Omron CX-Programmer project NewProject (CX-Programmer 9.81)

# PLC Sessao_10_02_2026_Exercicios: CP1L-E EM

## Global symbols (name address type ; comment)
0.00 BOOL  ; Interuptor 1
0.01 BOOL  ; Interruptor 2
0.02 BOOL  ; Botao de Emergencia
0.03 BOOL  ; Botao Stop
0.04 BOOL  ; Botao Start
0.05 BOOL  ; Botao Start 1
0.06 BOOL  ; Botao de Emergencia 2
0.07 BOOL  ; Botao Stop 1
0.08 BOOL  ; Flag do Temporizador 1
0.09 BOOL  ; Botao de Start Esquerdo
0.10 BOOL  ; Botao de Start Direito
0.11 BOOL  ; Temporizador
100 CHANNEL  ; Temporizador
100.00 BOOL  ; Lampada 1
100.01 BOOL  ; Lampada 2
100.02 BOOL  ; Lampada 3
100.03 BOOL  ; Lampada 4
100.04 BOOL  ; Bobina do Rele
100.05 BOOL  ; Bobina do Motor 1
100.06 BOOL  ; Bobina do Motor 2
100.07 BOOL  ; Temporizador
500 CHANNEL  ; Temporizador 1
T0001 BOOL  ; Flag do Temporizador 1

## Program NewProgram1 (cyclic task 0)
Local symbols
B_Emergencia 0.02 BOOL  ; Botao de emergencia
B_Rele 100.04 BOOL  ; Bobina do Rele
B_Start 0.04 BOOL  ; Botao Start
B_Stop 0.03 BOOL  ; Botao Stop
I_1 0.00 BOOL  ; Interruptor 1
I_2 0.01 BOOL  ; Interruptor 2
KM1 100.05 BOOL  ; Bobina do motor 1
KM2 100.06 BOOL  ; Bobina do motor 2
L_1 100.00 BOOL  ; Lampada 1
L_2 100.01 BOOL  ; Lampada 2
L_3 100.02 BOOL  ; Lampada 3
L_4 100.03 BOOL  ; Lampada 4

### Section Exercicio_1

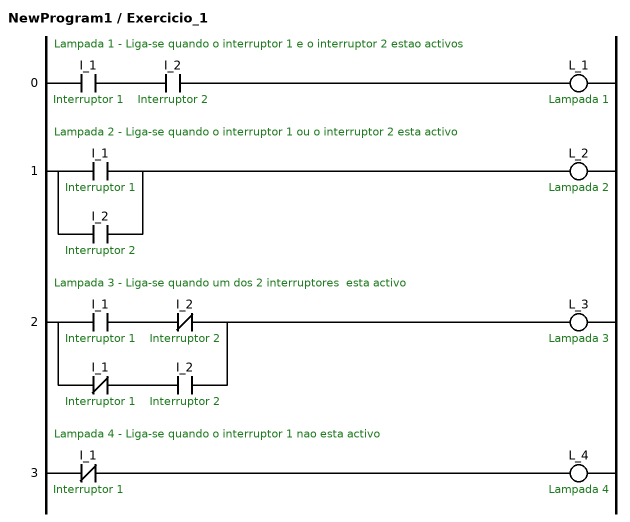
; rung 0: Lampada 1 - Liga-se quando o interruptor 1 e o interruptor 2 estao activos
LD I_1  ; Interruptor 1
AND I_2  ; Interruptor 2
OUT L_1  ; Lampada 1
; rung 1: Lampada 2 - Liga-se quando o interruptor 1 ou o interruptor 2 esta activo
LD I_1  ; Interruptor 1
OR I_2  ; Interruptor 2
OUT L_2  ; Lampada 2
; rung 2: Lampada 3 - Liga-se quando um dos 2 interruptores  esta activo
LD I_1  ; Interruptor 1
ANDNOT I_2  ; Interruptor 2
LDNOT I_1  ; Interruptor 1
AND I_2  ; Interruptor 2
ORLD
OUT L_3  ; Lampada 3
; rung 3: Lampada 4 - Liga-se quando o interruptor 1 nao esta activo
LDNOT I_1  ; Interruptor 1
OUT L_4  ; Lampada 4

### Section Exercicio_2

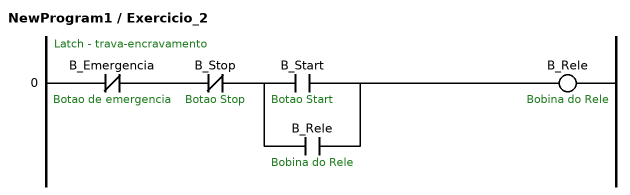
; rung 0: Latch - trava-encravamento
LDNOT B_Emergencia  ; Botao de emergencia
ANDNOT B_Stop  ; Botao Stop
LD B_Start  ; Botao Start
OR B_Rele  ; Bobina do Rele
ANDLD
OUT B_Rele  ; Bobina do Rele

### Section Exercicio_3

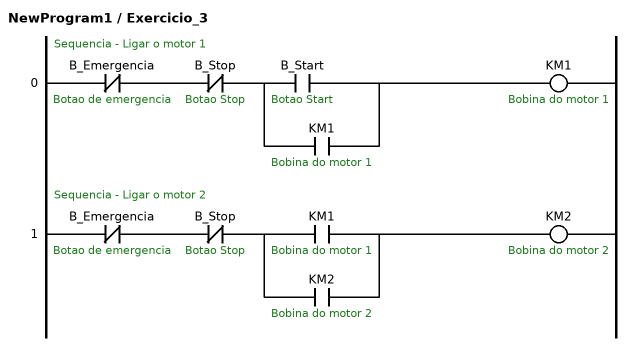
; rung 0: Sequencia - Ligar o motor 1
LDNOT B_Emergencia  ; Botao de emergencia
ANDNOT B_Stop  ; Botao Stop
LD B_Start  ; Botao Start
OR KM1  ; Bobina do motor 1
ANDLD
OUT KM1  ; Bobina do motor 1
; rung 1: Sequencia - Ligar o motor 2
LDNOT B_Emergencia  ; Botao de emergencia
ANDNOT B_Stop  ; Botao Stop
LD KM1  ; Bobina do motor 1
OR KM2  ; Bobina do motor 2
ANDLD
OUT KM2  ; Bobina do motor 2

### Section END
; rung 0
END(001)